FUNCTION INTERNAL Cbrt : LREAL
VAR_INPUT
  x : LREAL;
END_VAR
VAR
  xn : LREAL;
  h : LREAL;
END_VAR

Cbrt := SEL(x < 0, 1.0, -1.0) * EXPT(ABS(x), 1.0 / 3.0);

END_FUNCTION

(* stored: Version 1.1.0.1, ProductVersion 3.1.4024.9
   POU Cbrt: Id {e2df428d-5876-4ac5-a001-8b2714e1a509}, SpecialFunc None *)
